RoboDK station: RobotWorkstation.rdk

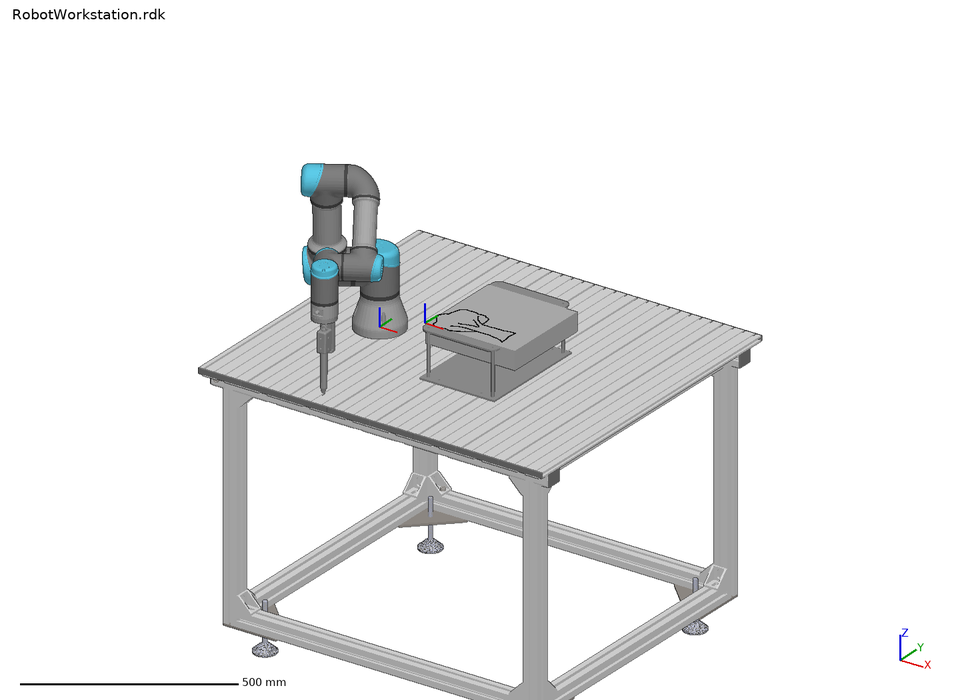
[picture v0: the station drawn from its stored meshes, robots at their saved joint values, targets as dots, program paths as lines]
Station 机器人绘图工作站. Poses are relative to the parent item; angles as X-Y-Z fixed-axis rotations.
  - object  at (0, 0, 0) mm, size 3 x 3 x 1 mm, geometry from .sld
  - object  at (0, 0, 0) mm, size 960 x 880 x 736.1 mm, geometry from .step
  - frame 绘图坐标系 at (200, -176.36, 13.37) mm
    - object  at (0.98, -0.26, 0) mm, size 250 x 250 x 50 mm, geometry from .sld
    - object  at (0.98, -0.26, 0) mm, size 203 x 115.1 x 51 mm, geometry from .sld
  - frame UR3 Base at (0, -72, -93) mm
    - robot UR3: 6 axes, payload 3 kg, reach 500 mm, repeatability 0.1 mm, weight 11 kg
        modified DH rows (alpha deg, a mm, theta deg, d mm): 0, 0, 0, 151.9; 90, 0, 180, 0; 0, 243.65, 0, 0; 0, 213, 0, 110.4; -90, 0, 0, 83.4; 90, 0, 180, 82.4
        joint limits [-360, -360, -360, -360, -360, -360] to [360, 360, 360, 360, 360, 360]; home [0, -90, -90, 0, 90, 0]; saved at [-58.314, -100.428, -121.765, -45.846, 89.752, 27.532]
      - tool , TCP at (0, 0, 170.9) mm, size 61 x 61 x 208 mm
  - object  at (200, -200, 10) mm, size 210.1 x 310.1 x 130 mm, geometry from .step
  - Python program simulate (listed below)

--- Python program simulate ---
from robolink import *      # 加载robolink模块
from robodk import *        # 加载robodk模块

import sys                  # 加载sys模块
import os                   # 加载os
import json
import time
import math

stroke_count = 0
RDK = Robolink(args='RobotWorkstation.rdk')            # 定义RoboDK工作站
#cam = camera.CameraModule(2)
path_stationfile = RDK.getParam('PATH_OPENSTATION')     # 获取当前工作站的路径
sys.path.append(os.path.abspath(path_stationfile))      # 将当前工作站的路径添加到系统路径中
from d import pen_track

# 定义工作站中的对象
robot = RDK.Item('UR3')            # 定义机器人对象
write_frame = RDK.Item('绘图坐标系')              # 定义写字坐标系：write_frame
write_tool = RDK.Item('书写工具')                    # 定义写字工具
pixel = RDK.Item('像素点')                        # 定义写字像素点
image_template = RDK.Item('模板')                 # 定义画板的模板
image = RDK.Item('画板')                          # 预定义工作站的画板

robot.setPoseFrame(write_frame)                              # 定义机器人的工件坐标系
robot.setPoseTool(write_tool)                                # 定义机器人的工具坐标系

######## 定义函数 ###########

# 定义函数：将二维空间中的点转化为三维空间中的点（4*4矩阵）
def point2D_2_pose(point, tangent):
    return transl(point.x, point.y, 0)*rotz(tangent.angle())

# s=0，笔从不接触纸面到接触纸面
def point2D_2_pose0(point, tangent):
    return transl(point.x, point.y, )*rotz(tangent.angle())

# s=1，接触保持纸面
def point2D_2_pose1(point, tangent):
    return transl(point.x, point.y, )*rotz(tangent.angle())

# s=2，从接触纸面到离开纸面
def point2D_2_pose2(point, tangent):
    return transl(point.x, point.y, )*rotz(tangent.angle())

def write_robot(list, item_frame, item_tool, robot):
    APPROACH = 70                                    # 定义常量APPROACH为100
    orient_frame2tool = roty(pi)
    global stroke_count
    x = None
    y = None
    for p in list:
        size = 150
        y = p[0]*size/1024
        x = size - p[1]*size/1024
        if p[3]==0 or p[3]==2:
            target0 = transl(x, y, 20)*orient_frame2tool         # 将p_0转化为机器人目标点target_0(4*4矩阵)
        elif p[3]==1:
            z = 20+(3.8-math.log(p[2]))*2-p[2]*0.3
            if z<0:
                z = 0
            target0=transl(x, y, z)*orient_frame2tool
        target0_app = target0*transl(0,0,-APPROACH)             # 定义目标点：target0_app
        print(str(target0_app))
#        raise Exception
        robot.MoveL(target0_app)
        if p[3]==2:
            stroke_count += 1
            print(stroke_count)

def dip(item_frame, item_tool, robot):
    home_joints = [-45,-90,-70,-90,90,0]
    APPROACH = 140
    orient_frame2tool = roty(pi)
    robot.MoveJ(home_joints)
    time.sleep(5)
    print('home_joints')

    # go down
    x = -150
    y = -200
    target = transl(x, y, -APPROACH)*orient_frame2tool
    robot.MoveL(target)

    # rotate
    target1 = transl(x+50, y+30, -APPROACH+10)*orient_frame2tool
    target1 = target1*rotz(1.0)
    robot.MoveL(target1)
    print(1)
    target2 = transl(x-50, y-20, -APPROACH+15)*orient_frame2tool
    robot.MoveL(target2)
    print(2)
    target3 = transl(x-50, y+20, -APPROACH+30)*orient_frame2tool
    target3 = target3*rotz(-1.0)
    robot.MoveL(target3)
    target4 = transl(x-50, y-10, -APPROACH+40)*orient_frame2tool
    robot.MoveL(target4)
    target5 = transl(x-10, y+10, -APPROACH+70)*orient_frame2tool
    target5 = target5*rotz(1.0)
    robot.MoveL(target5)
    print('end')
    target = transl(x-10, y, -APPROACH+300)*orient_frame2tool
    robot.MoveJ(target)
    time.sleep(2)
    robot.MoveJ(home_joints)
    time.sleep(5)
    print('home_joints')

    # lift
    #robot.MoveL(home_joints)



    # robot.MoveL(home_joints)

######## 机器人写字主程序 #########


#c = input('请输入对联：')

from flask import Flask, request, render_template
import requests
app = Flask(__name__)
robot_busy = False

@app.route('/')
def main():
    return '<p>Hello, World!<p>'

@app.route('/test')
def test():
    global robot_busy
    if robot_busy:
        return 'Robot is busy.'
    else:
        robot_busy = True
    couplet = '测试'
    for s in couplet:
        print(s)
        # json_path = os.path.join(path_stationfile,'characters_tracks.json')
        # with open(json_path,'r') as js:
            # track = json.load(js)
        # a = track[s]
        a = pen_track(s)
        a = [j for i in a for j in i]
        write_robot(a, write_frame, write_tool, robot)
    robot_busy = False
    return 'finished'

@app.route('/connect', methods=['GET',])
def connect():
    if RDK.RunMode() != RUNMODE_SIMULATE:
        return 'Already connected.'
    else:
        robot.setConnectionParams('192.168.1.2',2000,'/programs/', 'root','easybot')
        #robot.setConnectionParams('192.168.1.3',2000,)
        success = robot.Connect()
        status, status_msg = robot.ConnectedState()
        time.sleep(2)
        if status != ROBOTCOM_READY:
            # Stop if the connection did not succeed
            return status_msg
        else:
            RDK.setRunMode(RUNMODE_RUN_ROBOT)
            inititial()
            return success

@app.route('/init')
def inititial():
    home_joints = [-45,-90,-70,-90,90,0]                                # 定义机器人的起始位置
  # home_joints = [0,0,15,-90,90,0]
    robot.MoveJ(home_joints)
    return 'Success'

@app.route('/write/<c>')
def write(c):
    global robot_busy
    global stroke_count
    if robot_busy:
        return 'Robot is busy.'
    else:
        robot_busy = True
    dip1()
    for s in c:
        print('write',stroke_count)
        if stroke_count>=10:
            stroke_count = 0
            dip1()
        if s == " ":
            time.sleep(10)
            continue
        print(s)
        a = pen_track(s)
        if a is None:
            continue
        a = [j for i in a for j in i]
        write_robot(a, write_frame, write_tool, robot)
        time.sleep(2)
    robot_busy = False
    return 'finished'

@app.route('/couplet', methods=['GET'])
def couplet():
    data = request.values.to_dict()['c']
    r = requests.get(f'http://localhost:12345/{data}')
    if r.status_code == 200 and r.text != 'Failed':
        if write(data)=='Robot is busy.':
            return 'Robot is busy.'
        inititial()
        time.sleep(10)
        if write(r.text)=='Robot is busy.':
            return 'Robot is busy.'
    return finished

@app.route('/dip')
def dip1():
    print('dip')
    dip(write_frame, write_tool, robot)
    return '1'


@app.route('/ocr')
def ocr():
    global cam
    s = couplet_ocr.ocr_current_camera(cam)
    print(s)
    r = requests.get(f'http://localhost:12345/{s}')
    if r.status_code == 200 and r.text != 'Failed':
        result = r.text
        return render_template('./tem.html', s=s+' '+result)
    return r.text

if __name__ == '__main__':
    dip()
